Staubli VAL3: Trasladar.pjx

--- Trasladar.pjx ---
Parameters version=s7.10 stackSize=5000 millimeterUnit=true
Program file=_GLOBAL.pgx
Program file=_INFO.pgx
Program file=mcp.pgx
Program file=robot.pgx
Program file=start.pgx
Program file=stop.pgx
Data file=Trasladar.dtx

--- Trasladar.dtx ---
bool bTraslada
bool bFin
bool bPiezaPreparada
bool bTermina
jointRx jHome
public mdesc mNomSpeed = {leave=25, reach=25}
mdesc mVelAprox = {accel=25, vel=50, decel=25, blend=off}
num nPendientes
num nSolicitadas = 2
pointRx pEntrada = {x=-415, y=250, z=-265, ry=-180, shoulder=lefty, elbow=epositive, wrist=wpositive, fatherId=world[0]}
pointRx pEspera = {x=-415, y=250, z=-215, rx=-180, ry=-7.016709E-15, rz=-180, shoulder=lefty, elbow=epositive, wrist=wpositive, fatherId=world[0]}
pointRx pSalida = {x=-415, z=-210, ry=-180, fatherId=world[0]}
string sMensaje
tool tEyector = {z=22, fatherId=flange[0], ioLink=valve1, ioOpen=1, ioClose=1}
trsf trAprox = {z=-50}

--- start.pgx ---
program start()
begin
  // Se pone en marcha la aplicacion

  // Se establece el valor inicial de variables globales
  // BOOL
  bPiezaPreparada=false
  bFin=false
  bTermina=false
  bTraslada=false

  // NUM
  nSolicitadas=1
  nPendientes=0

  // STRING
  sMensaje=""

  // Se crean e inician las tareas de la aplicacion
  taskCreate "mcp",100,mcp()
  taskCreate "robot",100,robot()
end

--- _GLOBAL.pgx ---
program _GLOBAL()
begin
  // BOOL
  // - bFin: indicador de finalizacion de la tarea "robot".
  // - bPiezaPreparada: pieza preparada para ser trasladada.
  // - bTermina: orden de terminar la ejecucion de la aplicacion.
  // - bTraslada: orden de trasladar piezas.
  //
  // JOINT
  // - jHome: brazo en la posicion de referencia.
  //
  // MDESC
  // - mNomSpeed: descriptor de movimiento a velocidad nominal.
  // - mVelAprox: descriptor de movimiento a velocidad de aproximacion.
  //
  // NUM
  // - nPendientes: numero de piezas pendientes de trasladar.
  // - nSolicitadas: numero total de piezas a trasladar.
  //
  // POINT
  // - pEntrada: posicion de entrada (cogida) de las piezas.
  // - pEspera: posicion de reposo (esperando pieza preparada).
  // - pSalida: posicion de salida (suelta/colocacion) de las piezas.
  //
  // STRING
  // - sMensaje: mensaje para mostrar en la pantalla.
  //
  // TOOL
  // - tEyector: parametros de la herramienta (eyector de vacio con ventosas).
  //
  // TRSF
  // - trAprox: transformacion de aproximacion a las posiciones origen/destino.
end

--- _INFO.pgx ---
program _INFO()
begin
  // TRASLADAR (Nivel 1)
  //
  // Traslada un determinado numero de piezas de una posicion a otra.
  //
  // Version 0.0
  // copyright (c) 2022 victortorreslopez
  // GNU General Public License
  //
  // HISTORIAL DE VERSIONES
  // ----------------------
  // 0.0, 13/12/2022, VTL: Creacion (desde PickPlace, 2018)
  //
  // FUNCIONALIDAD
  // -------------
  // - F1: Traslada una cierta cantidad de piezas de una posicion a otra.
  // - F3: Edita el numero total de piezas a trasladar.
  // - F8: Sale de la aplicacion.
  //
  // SITUACION INICIAL
  // -----------------
  // - Brazo en su posicion de referencia.
  // - Una pieza en la posicion de entrada.
  // - Ninguna pieza en la posicion de salida.
  //
  // RECURSOS
  // --------
  // - Datos: BOOL, JOINT, MDESC, POINT, STRING, TOOL, TRSF.
  // - Instrucciones: title, userPage, while, cls, gotoxy, put, getKey, switch,
  //   appro, movej, waitEndMove, if, wait, movel, close, open, delay,
  //   taskCreate.
  //
  // NOTAS
  // -----
  // - Resuelto de la manera mas sencilla posible. Con el conjunto de
  //   instrucciones mas reducido y mas simple posible.
  // - El area de trabajo es una plataforma elevada a 100 mm del suelo.
  //
  // REFERENCIAS
  // -----------
  //
  // CELDA
  // -----
  // - Version: s7.10
  // - Tipo de robot: TX60
  // - Montaje: suelo
  // - Modo usrIn0: directo.
  //
  // DATOS
  // -----
  // - Plataforma = 400x300x3 mm
  // - Altura de la plataforma = 100 mm
  // - Pieza = 69x22x11 mm
  // - Herramienta (eyector) = 40.0x33.3x22.0 mm
end

--- initialize.pgx ---
program initialize()
begin
  // inicializa las variables globales
  //
  // copyright (c) 2018-2020 victortorreslopez
  //
  // GNU General Public License
  //
  // historial de modificaciones
  // - 0.1, 2020/11/20-18:30, VTL: actualizacion
  // - 0.0, 2018/10/14-11:01, VTL: creacion
  //
  // variables binarias
  bContinua=false
  bFin=false
  bSalir=false
  bTraslada=false

  // variables numericas
  nCV=0

  // cadenas de caracteres
  sMensaje=""
end

--- mcp.pgx ---
program mcp()
  local num nTecla
begin
  // Controla la pantalla del mando manual (MCP)
  //
  // Variables locales
  // - nTecla: codigo de la tecla pulsada

  // Se establece el titulo de la aplicacion
  title("TRASLADAR")

  // Se muestra en la pantalla la pagina de usuario principal
  userPage()

  // Bucle principal de la tarea
  while !bFin
    // Se borra la pantalla
    cls()

    // Se muestra informacion en la pantalla
    gotoxy(2,3)
    put("Total  = "+toString("4",nSolicitadas))
    gotoxy(2,4)
    put("Actual = "+toString("4",nPendientes))
    gotoxy(7,7)
    put(sMensaje)

    // Se muestran las etiquetas de las teclas de funcion
    gotoxy(0,13)
    put("Tra.")
    gotoxy(10,13)
    put("Tot.")
    gotoxy(35,13)
    put("Sal.")

    // Se procesa la tecla pulsada
    nTecla=getKey()
    switch nTecla
      // Enter - Orden de continuar
      case 270
        bPiezaPreparada=true
      break
      // F1 - Orden de trasladar piezas
      case 271
        bTraslada=true
      break
      // F3 - Orden de editar el numero de piezas a trasladar
      case 273
        gotoxy(14,3)
        get(nSolicitadas)
      break
      // F8 - Orden de salir de la aplicacion
      case 278
        bTermina=true
      break
    endSwitch

    // Se da paso a la siguiente tarea y se estabiliza la pantalla
    delay(0.1)
  endWhile
  bFin=false

  // Se muestra un mensaje de despedida
  cls()
  gotoxy(12,7)
  put("That's all folks")
end

--- robot.pgx ---
program robot()
  local pointRx pAprox
begin
  // Controla los movimientos del brazo
  //
  // Variables locales
  // - pAprox: punto de aproximacion

  // Se desplaza a la posicion de espera
  pEspera=appro(pEntrada,trAprox)
  movej(pEspera,tEyector,mNomSpeed)
  waitEndMove()

  // Bucle principal de la tarea
  while !bTermina
    if bTraslada
      for nPendientes=0 to nSolicitadas-1
        // Se espera la orden de pieza preparada para continuar
        sMensaje="pulse 'enter' para continuar"
        wait(bPiezaPreparada)
        bPiezaPreparada=false
        sMensaje=""

        // Se aproxima a la posicion de entrada (origen)
        pAprox=appro(pEntrada,trAprox)
        movej(pAprox,tEyector,mNomSpeed)
        // Se coje la pieza
        movel(pEntrada,tEyector,mVelAprox)
        close(tEyector)
        movel(pAprox,tEyector,mVelAprox)

        // Se aproxima a la posicion de salida (destino)
        pAprox=appro(pSalida,trAprox)
        movej(pAprox,tEyector,mNomSpeed)
        // Se suelta la pieza
        movel(pSalida,tEyector,mVelAprox)
        open(tEyector)
        movel(pAprox,tEyector,mVelAprox)

        // Se regresa a la posicion de espera
        movej(pEspera,tEyector,mNomSpeed)
        waitEndMove()
      endFor
      bTraslada=false
    endIf

    // Se da paso a la siguiente tarea
    delay(0)
  endWhile
  bTermina=false

  // Se regresa a la posicion de referencia
  movej(jHome,tEyector,mNomSpeed)
  waitEndMove()

  // Se informa de la finalizacion de la tarea
  bFin=true
end

--- robotMotion.pgx ---
program robotMotion()
  local pointRx pAprox
begin
  // Controla los movimientos del brazo
  //
  // copyright (c) 2018-2020 victortorreslopez
  //
  // GNU General Public License
  //
  // Variables locales
  // - pAprox: punto de aproximacion
  //
  // Historial de modificaciones
  // ---------------------------
  // 1.2, 2020/12/24, VTL: 2a revision general
  // 1.1, 2020/12/02, VTL: 1a revision
  // 0.0, 2018/10/14, VTL: creacion

  // Se desplaza a la posicion de reposo
  pReposo = appro(pOrigen, trAprox)
  movej(pReposo, tPinza, mNomSpeed)

  // Se abre la pinza
  waitEndMove()
  tPinza.gripper = true
  delay(tPinza.otime)

  // Bucle principal de la tarea
  while !bSalir
    if bTraslada
      for nCV = 0 to nPV-1
        // Se espera la orden de continuar
        sMensaje = "pulse 'enter' para continuar"
        wait(bContinua)
        bContinua = false
        sMensaje = ""

        // Se coge una pieza
        // Se aproxima a la posicion origen
        pAprox = appro(pOrigen, trAprox)
        movej(pAprox, tPinza, mNomSpeed)
        movel(pOrigen, tPinza, mVelAprox)
        // Se cierra la pinza
        waitEndMove()
        tPinza.gripper = false
        delay(tPinza.ctime)
        // Se aleja de la posicion origen
        movel(pAprox, tPinza, mVelAprox)

        // Se coloca una pieza
        // Se aproxima a la posicion destino
        pAprox = appro(pDestino, trAprox)
        movej(pAprox, tPinza, mNomSpeed)
        movel(pDestino, tPinza, mVelAprox)
        waitEndMove()
        // Se abre la pinza
        tPinza.gripper = true
        delay(tPinza.otime)
        // Se aleja de la posicion destino
        movel(pAprox, tPinza, mVelAprox)

        // Se regresa a la posicion de reposo
        movej(pReposo, tPinza, mNomSpeed)
      endFor
      waitEndMove()
      bTraslada = false
    endIf

    // Se da paso a la siguiente tarea
    delay(0)
  endWhile
  bSalir = false

  // Se regresa a la posicion de referencia
  movej(jHome,tPinza,mNomSpeed)

  // Se cierra la pinza
  waitEndMove()
  tPinza.gripper = false
  delay(tPinza.ctime)

  // Se informa de la finalizacion de la tarea
  bFin = true
end

--- stop.pgx ---
program stop()
begin
  // Se finaliza la aplicacion

  // Nada que hacer aqui!
end

--- userInterface.pgx ---
program userInterface()
  local num nTecla
begin
  // Controla la pantalla del mando manual (MCP)
  //
  // copyright (c) 2018-2020 victortorreslopez
  //
  // GNU General Public License
  //
  // Variables locales
  // - nTecla: codigo de la tecla pulsada
  //
  // Historial de modificaciones
  // ---------------------------
  // 1.2, 2020/12/24, VTL: 2a revision general
  // 1.1, 2020/12/02, VTL: 1a revision
  // 0.0, 2018/10/14, VTL: creacion

  // Se establece el titulo de la aplicacion
  title("PICK & PLACE")

  // Se establece la pagina de usuario en la pantalla
  userPage()

  // Bucle principal de la tarea
  while !bFin
    // Se borra la pantalla
    cls()

    // Se muestra informacion en la pantalla
    gotoxy(2, 3)
    put("Total   = " + toString("4", nPV))
    gotoxy(2, 4)
    put("Actual  = " + toString("4", nCV))
    gotoxy(7, 7)
    put(sMensaje)

    // Se muestran las etiquetas de las teclas de funcion
    gotoxy(0, 13)
    put("Tra.")
    gotoxy(10, 13)
    put("Tot.")
    gotoxy(35, 13)
    put("Sal.")

    // Se procesa la tecla pulsada
    nTecla = getKey()
    switch nTecla
      // Enter - Orden de continuar
      case 270
        bContinua = true
      break
      // F1 - Orden de trasladar piezas
      case 271
        bTraslada = true
      break
      // F3 - Orden de editar el numero de piezas a trasladar
      case 273
        gotoxy(15, 3)
        get(nPV)
      break
      // F8 - Orden de salir de la aplicacion
      case 278
        bSalir = true
      break
    endSwitch

    // Se da paso a la siguiente tarea y estabiliza la pantalla
    delay(0.1)
  endWhile
  bFin = false

  // Se muestra un mensaje de despedida
  cls()
  gotoxy(12, 7)
  put("That's all folks")
end
